                                        FB_Bacnet.StartStopCommand_139.bEnWrite := TRUE;
                                        FB_Bacnet.StartStopCommand_139.bVal := FALSE;
                                    13: 
                                        
                                        FB_Bacnet.StartStopCommand_140.bEnWrite := TRUE;
                                        FB_Bacnet.StartStopCommand_140.bVal := FALSE;
                                    14: 
                                        
                                        FB_Bacnet.StartStopCommand_141.bEnWrite := TRUE;
                                        FB_Bacnet.StartStopCommand_141.bVal := FALSE;
                                    15: 
                                        
                                        FB_Bacnet.StartStopCommand_142.bEnWrite := TRUE;
                                        FB_Bacnet.StartStopCommand_142.bVal := FALSE;
                                    16: 
                                        
                                        FB_Bacnet.StartStopCommand_143.bEnWrite := TRUE;
                                        FB_Bacnet.StartStopCommand_143.bVal := FALSE;
                                    17: 
                                        
                                        FB_Bacnet.StartStopCommand_144.bEnWrite := TRUE;
                                        FB_Bacnet.StartStopCommand_144.bVal := FALSE;
                                    18: 
                                        
                                        FB_Bacnet.StartStopCommand_145.bEnWrite := TRUE;
                                        FB_Bacnet.StartStopCommand_145.bVal := FALSE;
                                    19: 
                                        
                                        FB_Bacnet.StartStopCommand_146.bEnWrite := TRUE;
                                        FB_Bacnet.StartStopCommand_146.bVal := FALSE;
                                    20: 
                                        
                                        FB_Bacnet.StartStopCommand_147.bEnWrite := TRUE;
                                        FB_Bacnet.StartStopCommand_147.bVal := FALSE;
                                    21: 
                                        
                                        FB_Bacnet.StartStopCommand_148.bEnWrite := TRUE;
                                        FB_Bacnet.StartStopCommand_148.bVal := FALSE;
                                    22: 
                                        
                                        FB_Bacnet.StartStopCommand_149.bEnWrite := TRUE;
                                        FB_Bacnet.StartStopCommand_149.bVal := FALSE;
                                    23: 
                                        
                                        FB_Bacnet.StartStopCommand_226.bEnWrite := TRUE;
                                        FB_Bacnet.StartStopCommand_226.bVal := FALSE;
                                END_CASE
                            END_IF
                        END_FOR
                    END_IF
                END_IF
            END_IF

            // Weekend schedule
            IF currD = 0 OR currD = 6 THEN
                IF (wSchedWEHourStartF33_ <> wSchedWEHourEndF33_ OR wSchedWEMinStartF33_ <> wSchedWEMinEndF33_) THEN
                    // Schedule Unit ON
                    IF wSchedWEHourStartF33_ = currH AND wSchedWEMinStartF33_ = currM AND NOT bUnitTriggered THEN
                        bUnitTriggered := TRUE;
                        FOR i := 1 TO 23 DO
                            // Send command unit ON
                            IF bUnitF33_[i] THEN 
                                CASE i OF
                                    1: 
                                        
                                        FB_Bacnet.StartStopCommand_128.bEnWrite := TRUE;
                                        FB_Bacnet.StartStopCommand_128.bVal := TRUE;
                                    2: 
                                        
                                        FB_Bacnet.StartStopCommand_129.bEnWrite := TRUE;
                                        FB_Bacnet.StartStopCommand_129.bVal := TRUE;
                                    3: 
                                        
                                        FB_Bacnet.StartStopCommand_130.bEnWrite := TRUE;
                                        FB_Bacnet.StartStopCommand_130.bVal := TRUE;
                                    4: 
                                        
                                        FB_Bacnet.StartStopCommand_131.bEnWrite := TRUE;
                                        FB_Bacnet.StartStopCommand_131.bVal := TRUE;
                                    5: 
                                        
                                        FB_Bacnet.StartStopCommand_132.bEnWrite := TRUE;
                                        FB_Bacnet.StartStopCommand_132.bVal := TRUE;
                                    6: 
                                        
                                        FB_Bacnet.StartStopCommand_133.bEnWrite := TRUE;
                                        FB_Bacnet.StartStopCommand_133.bVal := TRUE;
                                    7: 
                                        
                                        FB_Bacnet.StartStopCommand_134.bEnWrite := TRUE;
                                        FB_Bacnet.StartStopCommand_134.bVal := TRUE;
                                    8: 
                                        
                                        FB_Bacnet.StartStopCommand_135.bEnWrite := TRUE;
                                        FB_Bacnet.StartStopCommand_135.bVal := TRUE;
                                    9: 
                                        
                                        FB_Bacnet.StartStopCommand_136.bEnWrite := TRUE;
                                        FB_Bacnet.StartStopCommand_136.bVal := TRUE;
                                    10: 
                                        
                                        FB_Bacnet.StartStopCommand_137.bEnWrite := TRUE;
                                        FB_Bacnet.StartStopCommand_137.bVal := TRUE;
                                    11: 
                                        
                                        FB_Bacnet.StartStopCommand_138.bEnWrite := TRUE;
                                        FB_Bacnet.StartStopCommand_138.bVal := TRUE;
                                    12: 
                                        
                                        FB_Bacnet.StartStopCommand_139.bEnWrite := TRUE;
                                        FB_Bacnet.StartStopCommand_139.bVal := TRUE;
                                    13: 
                                        
                                        FB_Bacnet.StartStopCommand_140.bEnWrite := TRUE;
                                        FB_Bacnet.StartStopCommand_140.bVal := TRUE;
                                    14: 
                                        
                                        FB_Bacnet.StartStopCommand_141.bEnWrite := TRUE;
                                        FB_Bacnet.StartStopCommand_141.bVal := TRUE;
                                    15: 
                                        
                                        FB_Bacnet.StartStopCommand_142.bEnWrite := TRUE;
                                        FB_Bacnet.StartStopCommand_142.bVal := TRUE;
                                    16: 
                                        
                                        FB_Bacnet.StartStopCommand_143.bEnWrite := TRUE;
                                        FB_Bacnet.StartStopCommand_143.bVal := TRUE;
                                    17: 
                                        
                                        FB_Bacnet.StartStopCommand_144.bEnWrite := TRUE;
                                        FB_Bacnet.StartStopCommand_144.bVal := TRUE;
                                    18: 
                                        
                                        FB_Bacnet.StartStopCommand_145.bEnWrite := TRUE;
                                        FB_Bacnet.StartStopCommand_145.bVal := TRUE;
                                    19: 
                                        
                                        FB_Bacnet.StartStopCommand_146.bEnWrite := TRUE;
                                        FB_Bacnet.StartStopCommand_146.bVal := TRUE;
                                    20: 
                                        
                                        FB_Bacnet.StartStopCommand_147.bEnWrite := TRUE;
                                        FB_Bacnet.StartStopCommand_147.bVal := TRUE;
                                    21: 
                                        
                                        FB_Bacnet.StartStopCommand_148.bEnWrite := TRUE;
                                        FB_Bacnet.StartStopCommand_148.bVal := TRUE;
                                    22: 
                                        
                                        FB_Bacnet.StartStopCommand_149.bEnWrite := TRUE;
                                        FB_Bacnet.StartStopCommand_149.bVal := TRUE;
                                    23: 
                                        
                                        FB_Bacnet.StartStopCommand_226.bEnWrite := TRUE;
                                        FB_Bacnet.StartStopCommand_226.bVal := TRUE;
                                END_CASE
                            END_IF
                        END_FOR
                    END_IF
                    // Schedule Unit OFF
                    IF wSchedWEHourEndF33_ = currH AND wSchedWEMinEndF33_ = currM AND NOT bUnitTriggered THEN
                        bUnitTriggered := TRUE;
                        FOR i := 1 TO 23 DO
                            // Send command unit OFF
                            IF bUnitF33_[i] THEN 
                                CASE i OF
                                    1: 
                                        
                                        FB_Bacnet.StartStopCommand_128.bEnWrite := TRUE;
                                        FB_Bacnet.StartStopCommand_128.bVal := FALSE;
                                    2: 
                                        
                                        FB_Bacnet.StartStopCommand_129.bEnWrite := TRUE;
                                        FB_Bacnet.StartStopCommand_129.bVal := FALSE;
                                    3: 
                                        
                                        FB_Bacnet.StartStopCommand_130.bEnWrite := TRUE;
                                        FB_Bacnet.StartStopCommand_130.bVal := FALSE;
                                    4: 
                                        
                                        FB_Bacnet.StartStopCommand_131.bEnWrite := TRUE;
                                        FB_Bacnet.StartStopCommand_131.bVal := FALSE;
                                    5: 
                                        
                                        FB_Bacnet.StartStopCommand_132.bEnWrite := TRUE;
                                        FB_Bacnet.StartStopCommand_132.bVal := FALSE;
                                    6: 
                                        
                                        FB_Bacnet.StartStopCommand_133.bEnWrite := TRUE;
                                        FB_Bacnet.StartStopCommand_133.bVal := FALSE;
                                    7: 
                                        
                                        FB_Bacnet.StartStopCommand_134.bEnWrite := TRUE;
                                        FB_Bacnet.StartStopCommand_134.bVal := FALSE;
                                    8: 
                                        
                                        FB_Bacnet.StartStopCommand_135.bEnWrite := TRUE;
                                        FB_Bacnet.StartStopCommand_135.bVal := FALSE;
                                    9: 
                                        
                                        FB_Bacnet.StartStopCommand_136.bEnWrite := TRUE;
                                        FB_Bacnet.StartStopCommand_136.bVal := FALSE;
                                    10: 
                                        
                                        FB_Bacnet.StartStopCommand_137.bEnWrite := TRUE;
                                        FB_Bacnet.StartStopCommand_137.bVal := FALSE;
                                    11: 
                                        
                                        FB_Bacnet.StartStopCommand_138.bEnWrite := TRUE;
                                        FB_Bacnet.StartStopCommand_138.bVal := FALSE;
                                    12: 
                                        
                                        FB_Bacnet.StartStopCommand_139.bEnWrite := TRUE;
                                        FB_Bacnet.StartStopCommand_139.bVal := FALSE;
                                    13: 
                                        
                                        FB_Bacnet.StartStopCommand_140.bEnWrite := TRUE;
                                        FB_Bacnet.StartStopCommand_140.bVal := FALSE;
                                    14: 
                                        
                                        FB_Bacnet.StartStopCommand_141.bEnWrite := TRUE;
                                        FB_Bacnet.StartStopCommand_141.bVal := FALSE;
                                    15: 
                                        
                                        FB_Bacnet.StartStopCommand_142.bEnWrite := TRUE;
                                        FB_Bacnet.StartStopCommand_142.bVal := FALSE;
                                    16: 
                                        
                                        FB_Bacnet.StartStopCommand_143.bEnWrite := TRUE;
                                        FB_Bacnet.StartStopCommand_143.bVal := FALSE;
                                    17: 
                                        
                                        FB_Bacnet.StartStopCommand_144.bEnWrite := TRUE;
                                        FB_Bacnet.StartStopCommand_144.bVal := FALSE;
                                    18: 
                                        
                                        FB_Bacnet.StartStopCommand_145.bEnWrite := TRUE;
                                        FB_Bacnet.StartStopCommand_145.bVal := FALSE;
                                    19: 
                                        
                                        FB_Bacnet.StartStopCommand_146.bEnWrite := TRUE;
                                        FB_Bacnet.StartStopCommand_146.bVal := FALSE;
                                    20: 
                                        
                                        FB_Bacnet.StartStopCommand_147.bEnWrite := TRUE;
                                        FB_Bacnet.StartStopCommand_147.bVal := FALSE;
                                    21: 
                                        
                                        FB_Bacnet.StartStopCommand_148.bEnWrite := TRUE;
                                        FB_Bacnet.StartStopCommand_148.bVal := FALSE;
                                    22: 
                                        
                                        FB_Bacnet.StartStopCommand_149.bEnWrite := TRUE;
                                        FB_Bacnet.StartStopCommand_149.bVal := FALSE;
                                    23: 
                                        
                                        FB_Bacnet.StartStopCommand_226.bEnWrite := TRUE;
                                        FB_Bacnet.StartStopCommand_226.bVal := FALSE;
                                END_CASE
                            END_IF
                        END_FOR
                    END_IF
                END_IF
            END_IF
        END_IF

END_FUNCTION_BLOCK

// ---- POUs/FB_Scheduler/FB_Scheduler_F35.TcPOU

    FUNCTION_BLOCK FB_Scheduler_F35
      VAR_INPUT
          currH : WORD;
          currM : WORD;
          currD : WORD;
      END_VAR
      VAR_IN_OUT
          FB_Bacnet : FB_BACnet_DAIKIN_MasterStation_III_No_8;
      END_VAR
      VAR
          i : INT;
          bUnitTriggered : BOOL := FALSE; // New flag to track execution
          prevMinute : WORD := 0;        // New variable to track the previous minute
      END_VAR
      VAR PERSISTENT
          //scheduler var
          bEnSchedF35_ : BOOL := FALSE;
          wSchedWDHourStartF35_ : WORD; 
          wSchedWDMinStartF35_ : WORD; 
          wSchedWEHourStartF35_ : WORD; 
          wSchedWEMinStartF35_ : WORD;
          wSchedWDHourEndF35_ : WORD;
          wSchedWDMinEndF35_ : WORD;
          wSchedWEHourEndF35_ : WORD;
          wSchedWEMinEndF35_ : WORD;
          //unit var
          bUnitF35_ : ARRAY [1..25] OF BOOL;
      END_VAR


// Reset trigger flag at minute change or at the exact scheduled time
IF currM <> prevMinute OR 
   (currH = wSchedWDHourStartF35_ AND currM = wSchedWDMinStartF35_) OR 
   (currH = wSchedWDHourEndF35_ AND currM = wSchedWDMinEndF35_) THEN
    bUnitTriggered := FALSE;
    prevMinute := currM;
END_IF

// Unit Schedule Enable
IF bEnSchedF35_ THEN
    // Weekday schedule
    IF currD >= 1 AND currD <= 5 THEN
        IF (wSchedWDHourStartF35_ <> wSchedWDHourEndF35_ OR wSchedWDMinStartF35_ <> wSchedWDMinEndF35_) THEN
            // Schedule Unit ON
            IF wSchedWDHourStartF35_ = currH AND wSchedWDMinStartF35_ = currM AND NOT bUnitTriggered THEN
                bUnitTriggered := TRUE;
                FOR i := 1 TO 25 DO
                    // Send command unit ON
                    IF bUnitF35_[i] THEN 
                        CASE i OF
                            1: 
                                FB_Bacnet.StartStopCommand_192.bEnWrite := TRUE;
                                FB_Bacnet.StartStopCommand_192.bVal := TRUE;
                            2: 
                                FB_Bacnet.StartStopCommand_193.bEnWrite := TRUE;
                                FB_Bacnet.StartStopCommand_193.bVal := TRUE;
                            3: 
                                FB_Bacnet.StartStopCommand_194.bEnWrite := TRUE;
                                FB_Bacnet.StartStopCommand_194.bVal := TRUE;
                            4: 
                                FB_Bacnet.StartStopCommand_195.bEnWrite := TRUE;
                                FB_Bacnet.StartStopCommand_195.bVal := TRUE;
                            5: 
                                FB_Bacnet.StartStopCommand_196.bEnWrite := TRUE;
                                FB_Bacnet.StartStopCommand_196.bVal := TRUE;
                            6: 
                                FB_Bacnet.StartStopCommand_197.bEnWrite := TRUE;
                                FB_Bacnet.StartStopCommand_197.bVal := TRUE;
                            7: 
                                FB_Bacnet.StartStopCommand_198.bEnWrite := TRUE;
                                FB_Bacnet.StartStopCommand_198.bVal := TRUE;
                            8: 
                                FB_Bacnet.StartStopCommand_199.bEnWrite := TRUE;
                                FB_Bacnet.StartStopCommand_199.bVal := TRUE;
                            9: 
                                FB_Bacnet.StartStopCommand_200.bEnWrite := TRUE;
                                FB_Bacnet.StartStopCommand_200.bVal := TRUE;
                            10: 
                                FB_Bacnet.StartStopCommand_201.bEnWrite := TRUE;
                                FB_Bacnet.StartStopCommand_201.bVal := TRUE;
                            11: 
                                FB_Bacnet.StartStopCommand_202.bEnWrite := TRUE;
                                FB_Bacnet.StartStopCommand_202.bVal := TRUE;
                            12: 
                                FB_Bacnet.StartStopCommand_203.bEnWrite := TRUE;
                                FB_Bacnet.StartStopCommand_203.bVal := TRUE;
                            13: 
                                FB_Bacnet.StartStopCommand_204.bEnWrite := TRUE;
                                FB_Bacnet.StartStopCommand_204.bVal := TRUE;
                            14: 
                                FB_Bacnet.StartStopCommand_205.bEnWrite := TRUE;
                                FB_Bacnet.StartStopCommand_205.bVal := TRUE;
                            15: 
                                FB_Bacnet.StartStopCommand_206.bEnWrite := TRUE;
                                FB_Bacnet.StartStopCommand_206.bVal := TRUE;
                            16: 
                                FB_Bacnet.StartStopCommand_207.bEnWrite := TRUE;
                                FB_Bacnet.StartStopCommand_207.bVal := TRUE;
                            17: 
                                FB_Bacnet.StartStopCommand_208.bEnWrite := TRUE;
                                FB_Bacnet.StartStopCommand_208.bVal := TRUE;
                            18: 
                                FB_Bacnet.StartStopCommand_209.bEnWrite := TRUE;
                                FB_Bacnet.StartStopCommand_209.bVal := TRUE;
                            19: 
                                FB_Bacnet.StartStopCommand_210.bEnWrite := TRUE;
                                FB_Bacnet.StartStopCommand_210.bVal := TRUE;
                            20: 
                                FB_Bacnet.StartStopCommand_211.bEnWrite := TRUE;
                                FB_Bacnet.StartStopCommand_211.bVal := TRUE;
                            21: 
                                FB_Bacnet.StartStopCommand_212.bEnWrite := TRUE;
                                FB_Bacnet.StartStopCommand_212.bVal := TRUE;
                            22: 
                                FB_Bacnet.StartStopCommand_213.bEnWrite := TRUE;
                                FB_Bacnet.StartStopCommand_213.bVal := TRUE;
                            23: 
                                //FB_Bacnet.StartStopCommand_242.bEnWrite := TRUE;
                                //FB_Bacnet.StartStopCommand_242.bVal := TRUE;
                            24: 
                                FB_Bacnet.StartStopCommand_243.bEnWrite := TRUE;
                                FB_Bacnet.StartStopCommand_243.bVal := TRUE;
                            25: 
                                FB_Bacnet.StartStopCommand_227.bEnWrite := TRUE;
                                FB_Bacnet.StartStopCommand_227.bVal := TRUE;
                        END_CASE
                    END_IF
                END_FOR
            END_IF
            // Schedule Unit OFF
            IF wSchedWDHourEndF35_ = currH AND wSchedWDMinEndF35_ = currM AND NOT bUnitTriggered THEN
                bUnitTriggered := TRUE;
                FOR i := 1 TO 25 DO
                    // Send command unit OFF
                    IF bUnitF35_[i] THEN 
                        CASE i OF
                            1: 
                                FB_Bacnet.StartStopCommand_192.bEnWrite := TRUE;
                                FB_Bacnet.StartStopCommand_192.bVal := FALSE;
                            2: 
                                FB_Bacnet.StartStopCommand_193.bEnWrite := TRUE;
                                FB_Bacnet.StartStopCommand_193.bVal := FALSE;
                            3: 
                                FB_Bacnet.StartStopCommand_194.bEnWrite := TRUE;
                                FB_Bacnet.StartStopCommand_194.bVal := FALSE;
                            4: 
                                FB_Bacnet.StartStopCommand_195.bEnWrite := TRUE;
                                FB_Bacnet.StartStopCommand_195.bVal := FALSE;
                            5: 
                                FB_Bacnet.StartStopCommand_196.bEnWrite := TRUE;
                                FB_Bacnet.StartStopCommand_196.bVal := FALSE;
                            6: 
                                FB_Bacnet.StartStopCommand_197.bEnWrite := TRUE;
                                FB_Bacnet.StartStopCommand_197.bVal := FALSE;
                            7: 
                                FB_Bacnet.StartStopCommand_198.bEnWrite := TRUE;
                                FB_Bacnet.StartStopCommand_198.bVal := FALSE;
                            8: 
                                FB_Bacnet.StartStopCommand_199.bEnWrite := TRUE;
                                FB_Bacnet.StartStopCommand_199.bVal := FALSE;
                            9: 
                                FB_Bacnet.StartStopCommand_200.bEnWrite := TRUE;
                                FB_Bacnet.StartStopCommand_200.bVal := FALSE;
                            10: 
                                FB_Bacnet.StartStopCommand_201.bEnWrite := TRUE;
                                FB_Bacnet.StartStopCommand_201.bVal := FALSE;
                            11: 
                                FB_Bacnet.StartStopCommand_202.bEnWrite := TRUE;
                                FB_Bacnet.StartStopCommand_202.bVal := FALSE;
                            12: 
                                FB_Bacnet.StartStopCommand_203.bEnWrite := TRUE;
                                FB_Bacnet.StartStopCommand_203.bVal := FALSE;
                            13: 
                                FB_Bacnet.StartStopCommand_204.bEnWrite := TRUE;
                                FB_Bacnet.StartStopCommand_204.bVal := FALSE;
                            14: 
                                FB_Bacnet.StartStopCommand_205.bEnWrite := TRUE;
                                FB_Bacnet.StartStopCommand_205.bVal := FALSE;
                            15: 
                                FB_Bacnet.StartStopCommand_206.bEnWrite := TRUE;
                                FB_Bacnet.StartStopCommand_206.bVal := FALSE;
                            16: 
                                FB_Bacnet.StartStopCommand_207.bEnWrite := TRUE;
                                FB_Bacnet.StartStopCommand_207.bVal := FALSE;
                            17: 
                                FB_Bacnet.StartStopCommand_208.bEnWrite := TRUE;
                                FB_Bacnet.StartStopCommand_208.bVal := FALSE;
                            18: 
                                FB_Bacnet.StartStopCommand_209.bEnWrite := TRUE;
                                FB_Bacnet.StartStopCommand_209.bVal := FALSE;
                            19: 
                                FB_Bacnet.StartStopCommand_210.bEnWrite := TRUE;
                                FB_Bacnet.StartStopCommand_210.bVal := FALSE;
                            20: 
                                FB_Bacnet.StartStopCommand_211.bEnWrite := TRUE;
                                FB_Bacnet.StartStopCommand_211.bVal := FALSE;
                            21: 
                                FB_Bacnet.StartStopCommand_212.bEnWrite := TRUE;
                                FB_Bacnet.StartStopCommand_212.bVal := FALSE;
                            22: 
                                FB_Bacnet.StartStopCommand_213.bEnWrite := TRUE;
                                FB_Bacnet.StartStopCommand_213.bVal := FALSE;
                            23: 
                                //FB_Bacnet.StartStopCommand_242.bEnWrite := TRUE;
                                //FB_Bacnet.StartStopCommand_242.bVal := FALSE;
                            24: 
                                FB_Bacnet.StartStopCommand_243.bEnWrite := TRUE;
                                FB_Bacnet.StartStopCommand_243.bVal := FALSE;
                            25: 
                                FB_Bacnet.StartStopCommand_227.bEnWrite := TRUE;
                                FB_Bacnet.StartStopCommand_227.bVal := FALSE;
                        END_CASE
                    END_IF
                END_FOR
            END_IF
        END_IF
    END_IF

    // Weekend schedule
    IF currD = 0 OR currD = 6 THEN
        IF (wSchedWEHourStartF35_ <> wSchedWEHourEndF35_ OR wSchedWEMinStartF35_ <> wSchedWEMinEndF35_) THEN
            // Schedule Unit ON
            IF wSchedWEHourStartF35_ = currH AND wSchedWEMinStartF35_ = currM AND NOT bUnitTriggered THEN
                bUnitTriggered := TRUE;
                FOR i := 1 TO 25 DO
                    // Send command unit ON
                    IF bUnitF35_[i] THEN 
                        CASE i OF
                            1: 
                                FB_Bacnet.StartStopCommand_192.bEnWrite := TRUE;
                                FB_Bacnet.StartStopCommand_192.bVal := TRUE;
                            2: 
                                FB_Bacnet.StartStopCommand_193.bEnWrite := TRUE;
                                FB_Bacnet.StartStopCommand_193.bVal := TRUE;
                            3: 
                                FB_Bacnet.StartStopCommand_194.bEnWrite := TRUE;
                                FB_Bacnet.StartStopCommand_194.bVal := TRUE;
                            4: 
                                FB_Bacnet.StartStopCommand_195.bEnWrite := TRUE;
                                FB_Bacnet.StartStopCommand_195.bVal := TRUE;
                            5: 
                                FB_Bacnet.StartStopCommand_196.bEnWrite := TRUE;
                                FB_Bacnet.StartStopCommand_196.bVal := TRUE;
                            6: 
                                FB_Bacnet.StartStopCommand_197.bEnWrite := TRUE;
                                FB_Bacnet.StartStopCommand_197.bVal := TRUE;
                            7: 
                                FB_Bacnet.StartStopCommand_198.bEnWrite := TRUE;
                                FB_Bacnet.StartStopCommand_198.bVal := TRUE;
                            8: 
                                FB_Bacnet.StartStopCommand_199.bEnWrite := TRUE;
                                FB_Bacnet.StartStopCommand_199.bVal := TRUE;
                            9: 
                                FB_Bacnet.StartStopCommand_200.bEnWrite := TRUE;
                                FB_Bacnet.StartStopCommand_200.bVal := TRUE;
                            10: 
                                FB_Bacnet.StartStopCommand_201.bEnWrite := TRUE;
                                FB_Bacnet.StartStopCommand_201.bVal := TRUE;
                            11: 
                                FB_Bacnet.StartStopCommand_202.bEnWrite := TRUE;
                                FB_Bacnet.StartStopCommand_202.bVal := TRUE;
                            12: 
                                FB_Bacnet.StartStopCommand_203.bEnWrite := TRUE;
                                FB_Bacnet.StartStopCommand_203.bVal := TRUE;
                            13: 
                                FB_Bacnet.StartStopCommand_204.bEnWrite := TRUE;
                                FB_Bacnet.StartStopCommand_204.bVal := TRUE;
                            14: 
                                FB_Bacnet.StartStopCommand_205.bEnWrite := TRUE;
                                FB_Bacnet.StartStopCommand_205.bVal := TRUE;
                            15: 
                                FB_Bacnet.StartStopCommand_206.bEnWrite := TRUE;
                                FB_Bacnet.StartStopCommand_206.bVal := TRUE;
                            16: 
                                FB_Bacnet.StartStopCommand_207.bEnWrite := TRUE;
                                FB_Bacnet.StartStopCommand_207.bVal := TRUE;
                            17: 
                                FB_Bacnet.StartStopCommand_208.bEnWrite := TRUE;
                                FB_Bacnet.StartStopCommand_208.bVal := TRUE;
                            18: 
                                FB_Bacnet.StartStopCommand_209.bEnWrite := TRUE;
                                FB_Bacnet.StartStopCommand_209.bVal := TRUE;
                            19: 
                                FB_Bacnet.StartStopCommand_210.bEnWrite := TRUE;
                                FB_Bacnet.StartStopCommand_210.bVal := TRUE;
                            20: 
                                FB_Bacnet.StartStopCommand_211.bEnWrite := TRUE;
                                FB_Bacnet.StartStopCommand_211.bVal := TRUE;
                            21: 
                                FB_Bacnet.StartStopCommand_212.bEnWrite := TRUE;
                                FB_Bacnet.StartStopCommand_212.bVal := TRUE;
                            22: 
                                FB_Bacnet.StartStopCommand_213.bEnWrite := TRUE;
                                FB_Bacnet.StartStopCommand_213.bVal := TRUE;
                            23: 
                                //FB_Bacnet.StartStopCommand_242.bEnWrite := TRUE;
                                //FB_Bacnet.StartStopCommand_242.bVal := TRUE;
                            24: 
                                FB_Bacnet.StartStopCommand_243.bEnWrite := TRUE;
                                FB_Bacnet.StartStopCommand_243.bVal := TRUE;
                            25: 
                                FB_Bacnet.StartStopCommand_227.bEnWrite := TRUE;
                                FB_Bacnet.StartStopCommand_227.bVal := TRUE;
                        END_CASE
                    END_IF
                END_FOR        
            END_IF
            // Schedule Unit OFF
            IF wSchedWEHourEndF35_ = currH AND wSchedWEMinEndF35_ = currM AND NOT bUnitTriggered THEN
                bUnitTriggered := TRUE;
                FOR i := 1 TO 25 DO
                    // Send command unit OFF
                    IF bUnitF35_[i] THEN 
                        CASE i OF
                            1: 
                                FB_Bacnet.StartStopCommand_192.bEnWrite := TRUE;
                                FB_Bacnet.StartStopCommand_192.bVal := FALSE;
                            2: 
                                FB_Bacnet.StartStopCommand_193.bEnWrite := TRUE;
                                FB_Bacnet.StartStopCommand_193.bVal := FALSE;
                            3: 
                                FB_Bacnet.StartStopCommand_194.bEnWrite := TRUE;
                                FB_Bacnet.StartStopCommand_194.bVal := FALSE;
                            4: 
                                FB_Bacnet.StartStopCommand_195.bEnWrite := TRUE;
                                FB_Bacnet.StartStopCommand_195.bVal := FALSE;
                            5: 
                                FB_Bacnet.StartStopCommand_196.bEnWrite := TRUE;
                                FB_Bacnet.StartStopCommand_196.bVal := FALSE;
                            6: 
                                FB_Bacnet.StartStopCommand_197.bEnWrite := TRUE;
                                FB_Bacnet.StartStopCommand_197.bVal := FALSE;
                            7: 
                                FB_Bacnet.StartStopCommand_198.bEnWrite := TRUE;
                                FB_Bacnet.StartStopCommand_198.bVal := FALSE;
                            8: 
                                FB_Bacnet.StartStopCommand_199.bEnWrite := TRUE;
                                FB_Bacnet.StartStopCommand_199.bVal := FALSE;
                            9: 
                                FB_Bacnet.StartStopCommand_200.bEnWrite := TRUE;
                                FB_Bacnet.StartStopCommand_200.bVal := FALSE;
                            10: 
                                FB_Bacnet.StartStopCommand_201.bEnWrite := TRUE;
                                FB_Bacnet.StartStopCommand_201.bVal := FALSE;
                            11: 
                                FB_Bacnet.StartStopCommand_202.bEnWrite := TRUE;
                                FB_Bacnet.StartStopCommand_202.bVal := FALSE;
                            12: 
                                FB_Bacnet.StartStopCommand_203.bEnWrite := TRUE;
                                FB_Bacnet.StartStopCommand_203.bVal := FALSE;
                            13: 
                                FB_Bacnet.StartStopCommand_204.bEnWrite := TRUE;
                                FB_Bacnet.StartStopCommand_204.bVal := FALSE;
                            14: 
                                FB_Bacnet.StartStopCommand_205.bEnWrite := TRUE;
                                FB_Bacnet.StartStopCommand_205.bVal := FALSE;
                            15: 
                                FB_Bacnet.StartStopCommand_206.bEnWrite := TRUE;
                                FB_Bacnet.StartStopCommand_206.bVal := FALSE;
                            16: 
                                FB_Bacnet.StartStopCommand_207.bEnWrite := TRUE;
                                FB_Bacnet.StartStopCommand_207.bVal := FALSE;
                            17: 
                                FB_Bacnet.StartStopCommand_208.bEnWrite := TRUE;
                                FB_Bacnet.StartStopCommand_208.bVal := FALSE;
                            18: 
                                FB_Bacnet.StartStopCommand_209.bEnWrite := TRUE;
                                FB_Bacnet.StartStopCommand_209.bVal := FALSE;
                            19: 
                                FB_Bacnet.StartStopCommand_210.bEnWrite := TRUE;
                                FB_Bacnet.StartStopCommand_210.bVal := FALSE;
                            20: 
                                FB_Bacnet.StartStopCommand_211.bEnWrite := TRUE;
                                FB_Bacnet.StartStopCommand_211.bVal := FALSE;
                            21: 
                                FB_Bacnet.StartStopCommand_212.bEnWrite := TRUE;
                                FB_Bacnet.StartStopCommand_212.bVal := FALSE;
                            22: 
                                FB_Bacnet.StartStopCommand_213.bEnWrite := TRUE;
                                FB_Bacnet.StartStopCommand_213.bVal := FALSE;
                            23: 
                                //FB_Bacnet.StartStopCommand_242.bEnWrite := TRUE;
                                //FB_Bacnet.StartStopCommand_242.bVal := FALSE;
                            24: 
                                FB_Bacnet.StartStopCommand_243.bEnWrite := TRUE;
                                FB_Bacnet.StartStopCommand_243.bVal := FALSE;
                            25: 
                                FB_Bacnet.StartStopCommand_227.bEnWrite := TRUE;
                                FB_Bacnet.StartStopCommand_227.bVal := FALSE;
                        END_CASE
                    END_IF
                END_FOR
            END_IF
        END_IF
    END_IF
END_IF

END_FUNCTION_BLOCK

// ---- POUs/FB_Scheduler/FB_Scheduler_F36.TcPOU

      FUNCTION_BLOCK FB_Scheduler_F36
      VAR_INPUT
          currH : WORD;
          currM : WORD;
          currD : WORD;
      END_VAR
      VAR_IN_OUT
          FB_Bacnet : FB_BACnet_DAIKIN_MasterStation_III_No_9;
      END_VAR
      VAR
          i : INT;
          bUnitTriggered : BOOL := FALSE; // New flag to track execution
          prevMinute : WORD := 0;        // New variable to track the previous minute
      END_VAR
      VAR PERSISTENT
          //scheduler var
          bEnSchedF36_ : BOOL := FALSE;
          wSchedWDHourStartF36_ : WORD; 
          wSchedWDMinStartF36_ : WORD; 
          wSchedWEHourStartF36_ : WORD; 
          wSchedWEMinStartF36_ : WORD;
          wSchedWDHourEndF36_ : WORD;
          wSchedWDMinEndF36_ : WORD;
          wSchedWEHourEndF36_ : WORD;
          wSchedWEMinEndF36_ : WORD;
          //unit var
          bUnitF36_ : ARRAY [1..23] OF BOOL;
      END_VAR


        // Reset trigger flag at minute change or at the exact scheduled time
        IF currM <> prevMinute OR 
           (currH = wSchedWDHourStartF36_ AND currM = wSchedWDMinStartF36_) OR 
           (currH = wSchedWDHourEndF36_ AND currM = wSchedWDMinEndF36_) THEN
            bUnitTriggered := FALSE;
            prevMinute := currM;
        END_IF

        // Unit Schedule Enable
        IF bEnSchedF36_ THEN
            // Weekday schedule
            IF currD >= 1 AND currD <= 5 THEN
                IF (wSchedWDHourStartF36_ <> wSchedWDHourEndF36_ OR wSchedWDMinStartF36_ <> wSchedWDMinEndF36_) THEN
                    // Schedule Unit ON
                    IF wSchedWDHourStartF36_ = currH AND wSchedWDMinStartF36_ = currM AND NOT bUnitTriggered THEN
                        bUnitTriggered := TRUE;
                        FOR i := 1 TO 23 DO
                            // Send command unit ON
                            IF bUnitF36_[i] THEN 
                                CASE i OF
                                    1: 
                                        
                                        FB_Bacnet.StartStopCommand_000.bEnWrite := TRUE;
                                        FB_Bacnet.StartStopCommand_000.bVal := TRUE;
                                    2: 
                                        
                                        FB_Bacnet.StartStopCommand_001.bEnWrite := TRUE;
                                        FB_Bacnet.StartStopCommand_001.bVal := TRUE;
                                    3: 
                                        
                                        FB_Bacnet.StartStopCommand_002.bEnWrite := TRUE;
                                        FB_Bacnet.StartStopCommand_002.bVal := TRUE;
                                    4: 
                                        
                                        FB_Bacnet.StartStopCommand_003.bEnWrite := TRUE;
                                        FB_Bacnet.StartStopCommand_003.bVal := TRUE;
                                    5: 
                                        
                                        FB_Bacnet.StartStopCommand_004.bEnWrite := TRUE;
                                        FB_Bacnet.StartStopCommand_004.bVal := TRUE;
                                    6: 
                                        
                                        FB_Bacnet.StartStopCommand_005.bEnWrite := TRUE;
                                        FB_Bacnet.StartStopCommand_005.bVal := TRUE;
                                    7: 
                                        
                                        FB_Bacnet.StartStopCommand_006.bEnWrite := TRUE;
                                        FB_Bacnet.StartStopCommand_006.bVal := TRUE;
                                    8: 
                                        
                                        FB_Bacnet.StartStopCommand_007.bEnWrite := TRUE;
                                        FB_Bacnet.StartStopCommand_007.bVal := TRUE;
                                    9: 
                                        
                                        FB_Bacnet.StartStopCommand_008.bEnWrite := TRUE;
                                        FB_Bacnet.StartStopCommand_008.bVal := TRUE;
                                    10: 
                                        
                                        FB_Bacnet.StartStopCommand_009.bEnWrite := TRUE;
                                        FB_Bacnet.StartStopCommand_009.bVal := TRUE;
                                    11: 
                                        
                                        FB_Bacnet.StartStopCommand_010.bEnWrite := TRUE;
                                        FB_Bacnet.StartStopCommand_010.bVal := TRUE;
                                    12: 
                                        
                                        FB_Bacnet.StartStopCommand_011.bEnWrite := TRUE;
                                        FB_Bacnet.StartStopCommand_011.bVal := TRUE;
                                    13: 
                                        
                                        FB_Bacnet.StartStopCommand_012.bEnWrite := TRUE;
                                        FB_Bacnet.StartStopCommand_012.bVal := TRUE;
                                    14: 
                                        
                                        FB_Bacnet.StartStopCommand_013.bEnWrite := TRUE;
                                        FB_Bacnet.StartStopCommand_013.bVal := TRUE;
                                    15: 
                                        
                                        FB_Bacnet.StartStopCommand_014.bEnWrite := TRUE;
                                        FB_Bacnet.StartStopCommand_014.bVal := TRUE;
                                    16: 
                                        
                                        FB_Bacnet.StartStopCommand_015.bEnWrite := TRUE;
                                        FB_Bacnet.StartStopCommand_015.bVal := TRUE;
                                    17: 
                                        
                                        FB_Bacnet.StartStopCommand_016.bEnWrite := TRUE;
                                        FB_Bacnet.StartStopCommand_016.bVal := TRUE;
                                    18: 
                                        
                                        FB_Bacnet.StartStopCommand_017.bEnWrite := TRUE;
                                        FB_Bacnet.StartStopCommand_017.bVal := TRUE;
                                    19: 
                                        
                                        FB_Bacnet.StartStopCommand_018.bEnWrite := TRUE;
                                        FB_Bacnet.StartStopCommand_018.bVal := TRUE;
                                    20: 
                                        
                                        FB_Bacnet.StartStopCommand_019.bEnWrite := TRUE;
                                        FB_Bacnet.StartStopCommand_019.bVal := TRUE;
                                    21: 
                                        
                                        FB_Bacnet.StartStopCommand_020.bEnWrite := TRUE;
                                        FB_Bacnet.StartStopCommand_020.bVal := TRUE;
                                    22: 
                                        
                                        FB_Bacnet.StartStopCommand_021.bEnWrite := TRUE;
                                        FB_Bacnet.StartStopCommand_021.bVal := TRUE;
                                    23: 
                                        
                                        FB_Bacnet.StartStopCommand_224.bEnWrite := TRUE;
                                        FB_Bacnet.StartStopCommand_224.bVal := TRUE;
                                END_CASE
                            END_IF
                        END_FOR
                    END_IF
                    // Schedule Unit OFF
                    IF wSchedWDHourEndF36_ = currH AND wSchedWDMinEndF36_ = currM AND NOT bUnitTriggered THEN
                        bUnitTriggered := TRUE;
                        FOR i := 1 TO 23 DO
                            // Send command unit OFF
                            IF bUnitF36_[i] THEN 
                                CASE i OF
                                    1: 
                                        
                                        FB_Bacnet.StartStopCommand_000.bEnWrite := TRUE;
                                        FB_Bacnet.StartStopCommand_000.bVal := FALSE;
                                    2: 
                                        
                                        FB_Bacnet.StartStopCommand_001.bEnWrite := TRUE;
                                        FB_Bacnet.StartStopCommand_001.bVal := FALSE;
                                    3: 
                                        
                                        FB_Bacnet.StartStopCommand_002.bEnWrite := TRUE;
                                        FB_Bacnet.StartStopCommand_002.bVal := FALSE;
                                    4: 
                                        
                                        FB_Bacnet.StartStopCommand_003.bEnWrite := TRUE;
                                        FB_Bacnet.StartStopCommand_003.bVal := FALSE;
                                    5: 
                                        
                                        FB_Bacnet.StartStopCommand_004.bEnWrite := TRUE;
                                        FB_Bacnet.StartStopCommand_004.bVal := FALSE;
                                    6: 
                                        
                                        FB_Bacnet.StartStopCommand_005.bEnWrite := TRUE;
                                        FB_Bacnet.StartStopCommand_005.bVal := FALSE;
                                    7: 
                                        
                                        FB_Bacnet.StartStopCommand_006.bEnWrite := TRUE;
                                        FB_Bacnet.StartStopCommand_006.bVal := FALSE;
                                    8: 
                                        
                                        FB_Bacnet.StartStopCommand_007.bEnWrite := TRUE;
                                        FB_Bacnet.StartStopCommand_007.bVal := FALSE;
                                    9: 
                                        
                                        FB_Bacnet.StartStopCommand_008.bEnWrite := TRUE;
                                        FB_Bacnet.StartStopCommand_008.bVal := FALSE;
                                    10: 
                                        
                                        FB_Bacnet.StartStopCommand_009.bEnWrite := TRUE;
                                        FB_Bacnet.StartStopCommand_009.bVal := FALSE;
                                    11: 
                                        
                                        FB_Bacnet.StartStopCommand_010.bEnWrite := TRUE;
                                        FB_Bacnet.StartStopCommand_010.bVal := FALSE;
                                    12: 
                                        
                                        FB_Bacnet.StartStopCommand_011.bEnWrite := TRUE;
                                        FB_Bacnet.StartStopCommand_011.bVal := FALSE;
                                    13: 
                                        
                                        FB_Bacnet.StartStopCommand_012.bEnWrite := TRUE;
                                        FB_Bacnet.StartStopCommand_012.bVal := FALSE;
                                    14: 
                                        
                                        FB_Bacnet.StartStopCommand_013.bEnWrite := TRUE;
                                        FB_Bacnet.StartStopCommand_013.bVal := FALSE;
                                    15: 
                                        
                                        FB_Bacnet.StartStopCommand_014.bEnWrite := TRUE;
                                        FB_Bacnet.StartStopCommand_014.bVal := FALSE;
                                    16: 
                                        
                                        FB_Bacnet.StartStopCommand_015.bEnWrite := TRUE;
                                        FB_Bacnet.StartStopCommand_015.bVal := FALSE;
                                    17: 
                                        
                                        FB_Bacnet.StartStopCommand_016.bEnWrite := TRUE;
                                        FB_Bacnet.StartStopCommand_016.bVal := FALSE;
                                    18: 
                                        
                                        FB_Bacnet.StartStopCommand_017.bEnWrite := TRUE;
                                        FB_Bacnet.StartStopCommand_017.bVal := FALSE;
                                    19: 
                                        
                                        FB_Bacnet.StartStopCommand_018.bEnWrite := TRUE;
                                        FB_Bacnet.StartStopCommand_018.bVal := FALSE;
                                    20: 
                                        
                                        FB_Bacnet.StartStopCommand_019.bEnWrite := TRUE;
                                        FB_Bacnet.StartStopCommand_019.bVal := FALSE;
                                    21: 
                                        
                                        FB_Bacnet.StartStopCommand_020.bEnWrite := TRUE;
                                        FB_Bacnet.StartStopCommand_020.bVal := FALSE;
                                    22: 
                                        
                                        FB_Bacnet.StartStopCommand_021.bEnWrite := TRUE;
                                        FB_Bacnet.StartStopCommand_021.bVal := FALSE;
                                    23: 
                                        
                                        FB_Bacnet.StartStopCommand_224.bEnWrite := TRUE;
                                        FB_Bacnet.StartStopCommand_224.bVal := FALSE;
                                END_CASE
                            END_IF
                        END_FOR
                    END_IF
                END_IF
            END_IF

            // Weekend schedule
            IF currD = 0 OR currD = 6 THEN
                IF (wSchedWEHourStartF36_ <> wSchedWEHourEndF36_ OR wSchedWEMinStartF36_ <> wSchedWEMinEndF36_) THEN
                    // Schedule Unit ON
                    IF wSchedWEHourStartF36_ = currH AND wSchedWEMinStartF36_ = currM AND NOT bUnitTriggered THEN
                        bUnitTriggered := TRUE;
                        FOR i := 1 TO 23 DO
                            // Send command unit ON
                            IF bUnitF36_[i] THEN 
                                CASE i OF
                                    1: 
                                        
                                        FB_Bacnet.StartStopCommand_000.bEnWrite := TRUE;
                                        FB_Bacnet.StartStopCommand_000.bVal := TRUE;
                                    2: 
                                        
                                        FB_Bacnet.StartStopCommand_001.bEnWrite := TRUE;
                                        FB_Bacnet.StartStopCommand_001.bVal := TRUE;
                                    3: 
                                        
                                        FB_Bacnet.StartStopCommand_002.bEnWrite := TRUE;
                                        FB_Bacnet.StartStopCommand_002.bVal := TRUE;
                                    4: 
                                        
                                        FB_Bacnet.StartStopCommand_003.bEnWrite := TRUE;
                                        FB_Bacnet.StartStopCommand_003.bVal := TRUE;
                                    5: 
                                        
                                        FB_Bacnet.StartStopCommand_004.bEnWrite := TRUE;
                                        FB_Bacnet.StartStopCommand_004.bVal := TRUE;
                                    6: 
                                        
                                        FB_Bacnet.StartStopCommand_005.bEnWrite := TRUE;
                                        FB_Bacnet.StartStopCommand_005.bVal := TRUE;
                                    7: 
                                        
                                        FB_Bacnet.StartStopCommand_006.bEnWrite := TRUE;
                                        FB_Bacnet.StartStopCommand_006.bVal := TRUE;
                                    8: 
                                        
                                        FB_Bacnet.StartStopCommand_007.bEnWrite := TRUE;
                                        FB_Bacnet.StartStopCommand_007.bVal := TRUE;
                                    9: 
                                        
                                        FB_Bacnet.StartStopCommand_008.bEnWrite := TRUE;
                                        FB_Bacnet.StartStopCommand_008.bVal := TRUE;
                                    10: 
                                        
                                        FB_Bacnet.StartStopCommand_009.bEnWrite := TRUE;
                                        FB_Bacnet.StartStopCommand_009.bVal := TRUE;
                                    11: 
                                        
                                        FB_Bacnet.StartStopCommand_010.bEnWrite := TRUE;
                                        FB_Bacnet.StartStopCommand_010.bVal := TRUE;
                                    12: 
                                        
                                        FB_Bacnet.StartStopCommand_011.bEnWrite := TRUE;
                                        FB_Bacnet.StartStopCommand_011.bVal := TRUE;
                                    13: 
                                        
                                        FB_Bacnet.StartStopCommand_012.bEnWrite := TRUE;
                                        FB_Bacnet.StartStopCommand_012.bVal := TRUE;
                                    14: 
                                        
                                        FB_Bacnet.StartStopCommand_013.bEnWrite := TRUE;
                                        FB_Bacnet.StartStopCommand_013.bVal := TRUE;
                                    15: 
                                        
                                        FB_Bacnet.StartStopCommand_014.bEnWrite := TRUE;
                                        FB_Bacnet.StartStopCommand_014.bVal := TRUE;
                                    16: 
                                        
                                        FB_Bacnet.StartStopCommand_015.bEnWrite := TRUE;
                                        FB_Bacnet.StartStopCommand_015.bVal := TRUE;
                                    17: 
                                        
                                        FB_Bacnet.StartStopCommand_016.bEnWrite := TRUE;
                                        FB_Bacnet.StartStopCommand_016.bVal := TRUE;
                                    18: 
                                        
                                        FB_Bacnet.StartStopCommand_017.bEnWrite := TRUE;
                                        FB_Bacnet.StartStopCommand_017.bVal := TRUE;
                                    19: 
                                        
                                        FB_Bacnet.StartStopCommand_018.bEnWrite := TRUE;
                                        FB_Bacnet.StartStopCommand_018.bVal := TRUE;
                                    20: 
                                        
                                        FB_Bacnet.StartStopCommand_019.bEnWrite := TRUE;
                                        FB_Bacnet.StartStopCommand_019.bVal := TRUE;
                                    21: 
                                        
                                        FB_Bacnet.StartStopCommand_020.bEnWrite := TRUE;
                                        FB_Bacnet.StartStopCommand_020.bVal := TRUE;
                                    22: 
                                        
                                        FB_Bacnet.StartStopCommand_021.bEnWrite := TRUE;
                                        FB_Bacnet.StartStopCommand_021.bVal := TRUE;
                                    23: 
                                        
                                        FB_Bacnet.StartStopCommand_224.bEnWrite := TRUE;
                                        FB_Bacnet.StartStopCommand_224.bVal := TRUE;
                                END_CASE
                            END_IF
                        END_FOR
                    END_IF
                    // Schedule Unit OFF
                    IF wSchedWEHourEndF36_ = currH AND wSchedWEMinEndF36_ = currM AND NOT bUnitTriggered THEN
                        bUnitTriggered := TRUE;
                        FOR i := 1 TO 23 DO
                            // Send command unit OFF
                            IF bUnitF36_[i] THEN 
                                CASE i OF
                                    1: 
                                        
                                        FB_Bacnet.StartStopCommand_000.bEnWrite := TRUE;
                                        FB_Bacnet.StartStopCommand_000.bVal := FALSE;
                                    2: 
                                        
                                        FB_Bacnet.StartStopCommand_001.bEnWrite := TRUE;
                                        FB_Bacnet.StartStopCommand_001.bVal := FALSE;
                                    3: 
                                        
                                        FB_Bacnet.StartStopCommand_002.bEnWrite := TRUE;
                                        FB_Bacnet.StartStopCommand_002.bVal := FALSE;
                                    4: 
                                        
                                        FB_Bacnet.StartStopCommand_003.bEnWrite := TRUE;
                                        FB_Bacnet.StartStopCommand_003.bVal := FALSE;
                                    5: 
                                        
                                        FB_Bacnet.StartStopCommand_004.bEnWrite := TRUE;
                                        FB_Bacnet.StartStopCommand_004.bVal := FALSE;
                                    6: 
                                        
                                        FB_Bacnet.StartStopCommand_005.bEnWrite := TRUE;
                                        FB_Bacnet.StartStopCommand_005.bVal := FALSE;
                                    7: 
                                        
                                        FB_Bacnet.StartStopCommand_006.bEnWrite := TRUE;
                                        FB_Bacnet.StartStopCommand_006.bVal := FALSE;
                                    8: 
                                        
                                        FB_Bacnet.StartStopCommand_007.bEnWrite := TRUE;
                                        FB_Bacnet.StartStopCommand_007.bVal := FALSE;
                                    9: 
                                        
                                        FB_Bacnet.StartStopCommand_008.bEnWrite := TRUE;
                                        FB_Bacnet.StartStopCommand_008.bVal := FALSE;
                                    10: 
                                        
                                        FB_Bacnet.StartStopCommand_009.bEnWrite := TRUE;
                                        FB_Bacnet.StartStopCommand_009.bVal := FALSE;
                                    11: 
                                        
                                        FB_Bacnet.StartStopCommand_010.bEnWrite := TRUE;
                                        FB_Bacnet.StartStopCommand_010.bVal := FALSE;
                                    12: 
                                        
                                        FB_Bacnet.StartStopCommand_011.bEnWrite := TRUE;
                                        FB_Bacnet.StartStopCommand_011.bVal := FALSE;
                                    13: 
                                        
                                        FB_Bacnet.StartStopCommand_012.bEnWrite := TRUE;
                                        FB_Bacnet.StartStopCommand_012.bVal := FALSE;
                                    14: 
                                        
                                        FB_Bacnet.StartStopCommand_013.bEnWrite := TRUE;
                                        FB_Bacnet.StartStopCommand_013.bVal := FALSE;
                                    15: 
                                        
                                        FB_Bacnet.StartStopCommand_014.bEnWrite := TRUE;
                                        FB_Bacnet.StartStopCommand_014.bVal := FALSE;
                                    16: 
                                        
                                        FB_Bacnet.StartStopCommand_015.bEnWrite := TRUE;
                                        FB_Bacnet.StartStopCommand_015.bVal := FALSE;
                                    17: 
                                        
                                        FB_Bacnet.StartStopCommand_016.bEnWrite := TRUE;
                                        FB_Bacnet.StartStopCommand_016.bVal := FALSE;
                                    18: 
                                        
                                        FB_Bacnet.StartStopCommand_017.bEnWrite := TRUE;
                                        FB_Bacnet.StartStopCommand_017.bVal := FALSE;
                                    19: 
                                        
                                        FB_Bacnet.StartStopCommand_018.bEnWrite := TRUE;
                                        FB_Bacnet.StartStopCommand_018.bVal := FALSE;
                                    20: 
                                        
                                        FB_Bacnet.StartStopCommand_019.bEnWrite := TRUE;
                                        FB_Bacnet.StartStopCommand_019.bVal := FALSE;
                                    21: 
                                        
                                        FB_Bacnet.StartStopCommand_020.bEnWrite := TRUE;
                                        FB_Bacnet.StartStopCommand_020.bVal := FALSE;
                                    22: 
                                        
                                        FB_Bacnet.StartStopCommand_021.bEnWrite := TRUE;
                                        FB_Bacnet.StartStopCommand_021.bVal := FALSE;
                                    23: 
                                        
                                        FB_Bacnet.StartStopCommand_224.bEnWrite := TRUE;
                                        FB_Bacnet.StartStopCommand_224.bVal := FALSE;
                                END_CASE
                            END_IF
                        END_FOR
                    END_IF
                END_IF
            END_IF
        END_IF

END_FUNCTION_BLOCK

// ---- POUs/FB_Scheduler/FB_Scheduler_F37.TcPOU

      FUNCTION_BLOCK FB_Scheduler_F37
      VAR_INPUT
          currH : WORD;
          currM : WORD;
          currD : WORD;
      END_VAR
      VAR_IN_OUT
          FB_Bacnet : FB_BACnet_DAIKIN_MasterStation_III_No_9;
      END_VAR
      VAR
          i : INT;
          bUnitTriggered : BOOL := FALSE; // New flag to track execution
          prevMinute : WORD := 0;        // New variable to track the previous minute
      END_VAR
      VAR PERSISTENT
          //scheduler var
          bEnSchedF37_ : BOOL := FALSE;
          wSchedWDHourStartF37_ : WORD; 
          wSchedWDMinStartF37_ : WORD; 
          wSchedWEHourStartF37_ : WORD; 
          wSchedWEMinStartF37_ : WORD;
          wSchedWDHourEndF37_ : WORD;
          wSchedWDMinEndF37_ : WORD;
          wSchedWEHourEndF37_ : WORD;
          wSchedWEMinEndF37_ : WORD;
          //unit var
          bUnitF37_ : ARRAY [1..23] OF BOOL;
      END_VAR


        // Reset trigger flag at minute change or at the exact scheduled time
        IF currM <> prevMinute OR 
           (currH = wSchedWDHourStartF37_ AND currM = wSchedWDMinStartF37_) OR 
           (currH = wSchedWDHourEndF37_ AND currM = wSchedWDMinEndF37_) THEN
            bUnitTriggered := FALSE;
            prevMinute := currM;
        END_IF

        // Unit Schedule Enable
        IF bEnSchedF37_ THEN
            // Weekday schedule
            IF currD >= 1 AND currD <= 5 THEN
                IF (wSchedWDHourStartF37_ <> wSchedWDHourEndF37_ OR wSchedWDMinStartF37_ <> wSchedWDMinEndF37_) THEN
                    // Schedule Unit ON
                    IF wSchedWDHourStartF37_ = currH AND wSchedWDMinStartF37_ = currM AND NOT bUnitTriggered THEN
                        bUnitTriggered := TRUE;
                        FOR i := 1 TO 23 DO
                            // Send command unit ON
                            IF bUnitF37_[i] THEN 
                                CASE i OF
                                    1: 
                                        
                                        FB_Bacnet.StartStopCommand_064.bEnWrite := TRUE;
                                        FB_Bacnet.StartStopCommand_064.bVal := TRUE;
                                    2: 
                                        
                                        FB_Bacnet.StartStopCommand_065.bEnWrite := TRUE;
                                        FB_Bacnet.StartStopCommand_065.bVal := TRUE;
                                    3: 
                                        
                                        FB_Bacnet.StartStopCommand_066.bEnWrite := TRUE;
                                        FB_Bacnet.StartStopCommand_066.bVal := TRUE;
                                    4: 
                                        
                                        FB_Bacnet.StartStopCommand_067.bEnWrite := TRUE;
                                        FB_Bacnet.StartStopCommand_067.bVal := TRUE;
                                    5: 
                                        
                                        FB_Bacnet.StartStopCommand_068.bEnWrite := TRUE;
                                        FB_Bacnet.StartStopCommand_068.bVal := TRUE;
                                    6: 
                                        
                                        FB_Bacnet.StartStopCommand_069.bEnWrite := TRUE;
                                        FB_Bacnet.StartStopCommand_069.bVal := TRUE;
                                    7: 
                                        
                                        FB_Bacnet.StartStopCommand_070.bEnWrite := TRUE;
                                        FB_Bacnet.StartStopCommand_070.bVal := TRUE;
                                    8: 
                                        
                                        FB_Bacnet.StartStopCommand_071.bEnWrite := TRUE;
                                        FB_Bacnet.StartStopCommand_071.bVal := TRUE;
                                    9: 
                                        
                                        FB_Bacnet.StartStopCommand_072.bEnWrite := TRUE;
                                        FB_Bacnet.StartStopCommand_072.bVal := TRUE;
                                    10: 
                                        
                                        FB_Bacnet.StartStopCommand_073.bEnWrite := TRUE;
                                        FB_Bacnet.StartStopCommand_073.bVal := TRUE;
                                    11: 
                                        
                                        FB_Bacnet.StartStopCommand_074.bEnWrite := TRUE;
                                        FB_Bacnet.StartStopCommand_074.bVal := TRUE;
                                    12: 
                                        
                                        FB_Bacnet.StartStopCommand_075.bEnWrite := TRUE;
                                        FB_Bacnet.StartStopCommand_075.bVal := TRUE;
                                    13: 
                                        
                                        FB_Bacnet.StartStopCommand_076.bEnWrite := TRUE;
                                        FB_Bacnet.StartStopCommand_076.bVal := TRUE;
                                    14: 
                                        
                                        FB_Bacnet.StartStopCommand_077.bEnWrite := TRUE;
                                        FB_Bacnet.StartStopCommand_077.bVal := TRUE;
                                    15: 
                                        
                                        FB_Bacnet.StartStopCommand_078.bEnWrite := TRUE;
                                        FB_Bacnet.StartStopCommand_078.bVal := TRUE;
                                    16: 
                                        
                                        FB_Bacnet.StartStopCommand_079.bEnWrite := TRUE;
                                        FB_Bacnet.StartStopCommand_079.bVal := TRUE;
                                    17: 
                                        
                                        FB_Bacnet.StartStopCommand_080.bEnWrite := TRUE;
                                        FB_Bacnet.StartStopCommand_080.bVal := TRUE;
                                    18: 
                                        
                                        FB_Bacnet.StartStopCommand_081.bEnWrite := TRUE;
                                        FB_Bacnet.StartStopCommand_081.bVal := TRUE;
                                    19: 
                                        
                                        FB_Bacnet.StartStopCommand_082.bEnWrite := TRUE;
                                        FB_Bacnet.StartStopCommand_082.bVal := TRUE;
                                    20: 
                                        
                                        FB_Bacnet.StartStopCommand_083.bEnWrite := TRUE;
                                        FB_Bacnet.StartStopCommand_083.bVal := TRUE;
                                    21: 
                                        
                                        FB_Bacnet.StartStopCommand_084.bEnWrite := TRUE;
                                        FB_Bacnet.StartStopCommand_084.bVal := TRUE;
                                    22: 
                                        
                                        FB_Bacnet.StartStopCommand_085.bEnWrite := TRUE;
                                        FB_Bacnet.StartStopCommand_085.bVal := TRUE;
                                    23: 
                                        
                                        FB_Bacnet.StartStopCommand_225.bEnWrite := TRUE;
                                        FB_Bacnet.StartStopCommand_225.bVal := TRUE;
                                END_CASE
                            END_IF
                        END_FOR
                    END_IF
                    // Schedule Unit OFF
                    IF wSchedWDHourEndF37_ = currH AND wSchedWDMinEndF37_ = currM AND NOT bUnitTriggered THEN
                        bUnitTriggered := TRUE;
                        FOR i := 1 TO 23 DO
                            // Send command unit OFF
                            IF bUnitF37_[i] THEN 
                                CASE i OF
                                    1: 
                                        
                                        FB_Bacnet.StartStopCommand_064.bEnWrite := TRUE;
                                        FB_Bacnet.StartStopCommand_064.bVal := FALSE;
                                    2: 
                                        
                                        FB_Bacnet.StartStopCommand_065.bEnWrite := TRUE;
                                        FB_Bacnet.StartStopCommand_065.bVal := FALSE;
                                    3: 
                                        
                                        FB_Bacnet.StartStopCommand_066.bEnWrite := TRUE;
                                        FB_Bacnet.StartStopCommand_066.bVal := FALSE;
                                    4: 
                                        
                                        FB_Bacnet.StartStopCommand_067.bEnWrite := TRUE;
                                        FB_Bacnet.StartStopCommand_067.bVal := FALSE;
                                    5: 
                                        
                                        FB_Bacnet.StartStopCommand_068.bEnWrite := TRUE;
                                        FB_Bacnet.StartStopCommand_068.bVal := FALSE;
                                    6: 
                                        
                                        FB_Bacnet.StartStopCommand_069.bEnWrite := TRUE;
                                        FB_Bacnet.StartStopCommand_069.bVal := FALSE;
                                    7: 
                                        
                                        FB_Bacnet.StartStopCommand_070.bEnWrite := TRUE;
                                        FB_Bacnet.StartStopCommand_070.bVal := FALSE;
                                    8: 
                                        
                                        FB_Bacnet.StartStopCommand_071.bEnWrite := TRUE;
                                        FB_Bacnet.StartStopCommand_071.bVal := FALSE;
                                    9: 
                                        
                                        FB_Bacnet.StartStopCommand_072.bEnWrite := TRUE;
                                        FB_Bacnet.StartStopCommand_072.bVal := FALSE;
                                    10: 
                                        
                                        FB_Bacnet.StartStopCommand_073.bEnWrite := TRUE;
                                        FB_Bacnet.StartStopCommand_073.bVal := FALSE;
                                    11: 
                                        
                                        FB_Bacnet.StartStopCommand_074.bEnWrite := TRUE;
                                        FB_Bacnet.StartStopCommand_074.bVal := FALSE;
                                    12: 
                                        
                                        FB_Bacnet.StartStopCommand_075.bEnWrite := TRUE;
                                        FB_Bacnet.StartStopCommand_075.bVal := FALSE;
                                    13: 
                                        
                                        FB_Bacnet.StartStopCommand_076.bEnWrite := TRUE;
                                        FB_Bacnet.StartStopCommand_076.bVal := FALSE;
                                    14: 
                                        
                                        FB_Bacnet.StartStopCommand_077.bEnWrite := TRUE;
                                        FB_Bacnet.StartStopCommand_077.bVal := FALSE;
                                    15: 
                                        
                                        FB_Bacnet.StartStopCommand_078.bEnWrite := TRUE;
                                        FB_Bacnet.StartStopCommand_078.bVal := FALSE;
                                    16: 
                                        
                                        FB_Bacnet.StartStopCommand_079.bEnWrite := TRUE;
                                        FB_Bacnet.StartStopCommand_079.bVal := FALSE;
                                    17: 
                                        
                                        FB_Bacnet.StartStopCommand_080.bEnWrite := TRUE;
                                        FB_Bacnet.StartStopCommand_080.bVal := FALSE;
                                    18: 
                                        
                                        FB_Bacnet.StartStopCommand_081.bEnWrite := TRUE;
                                        FB_Bacnet.StartStopCommand_081.bVal := FALSE;
                                    19: 
                                        
                                        FB_Bacnet.StartStopCommand_082.bEnWrite := TRUE;
                                        FB_Bacnet.StartStopCommand_082.bVal := FALSE;
                                    20: 
                                        
                                        FB_Bacnet.StartStopCommand_083.bEnWrite := TRUE;
                                        FB_Bacnet.StartStopCommand_083.bVal := FALSE;
                                    21: 
                                        
                                        FB_Bacnet.StartStopCommand_084.bEnWrite := TRUE;
                                        FB_Bacnet.StartStopCommand_084.bVal := FALSE;
                                    22: 
                                        
                                        FB_Bacnet.StartStopCommand_085.bEnWrite := TRUE;
                                        FB_Bacnet.StartStopCommand_085.bVal := FALSE;
                                    23: 
                                        
                                        FB_Bacnet.StartStopCommand_225.bEnWrite := TRUE;
                                        FB_Bacnet.StartStopCommand_225.bVal := FALSE;
                                END_CASE
                            END_IF
                        END_FOR
                    END_IF
                END_IF
            END_IF

            // Weekend schedule
            IF currD = 0 OR currD = 6 THEN
                IF (wSchedWEHourStartF37_ <> wSchedWEHourEndF37_ OR wSchedWEMinStartF37_ <> wSchedWEMinEndF37_) THEN
                    // Schedule Unit ON
                    IF wSchedWEHourStartF37_ = currH AND wSchedWEMinStartF37_ = currM AND NOT bUnitTriggered THEN
                        bUnitTriggered := TRUE;
                        FOR i := 1 TO 23 DO
                            // Send command unit ON
                            IF bUnitF37_[i] THEN 
                                CASE i OF
                                    1: 
                                        
                                        FB_Bacnet.StartStopCommand_064.bEnWrite := TRUE;
                                        FB_Bacnet.StartStopCommand_064.bVal := TRUE;
                                    2: 
                                        
                                        FB_Bacnet.StartStopCommand_065.bEnWrite := TRUE;
                                        FB_Bacnet.StartStopCommand_065.bVal := TRUE;
                                    3: 
                                        
                                        FB_Bacnet.StartStopCommand_066.bEnWrite := TRUE;
                                        FB_Bacnet.StartStopCommand_066.bVal := TRUE;
                                    4: 
                                        
                                        FB_Bacnet.StartStopCommand_067.bEnWrite := TRUE;
                                        FB_Bacnet.StartStopCommand_067.bVal := TRUE;
                                    5: 
                                        
                                        FB_Bacnet.StartStopCommand_068.bEnWrite := TRUE;
                                        FB_Bacnet.StartStopCommand_068.bVal := TRUE;
                                    6: 
                                        
                                        FB_Bacnet.StartStopCommand_069.bEnWrite := TRUE;
                                        FB_Bacnet.StartStopCommand_069.bVal := TRUE;
                                    7: 
                                        
                                        FB_Bacnet.StartStopCommand_070.bEnWrite := TRUE;
                                        FB_Bacnet.StartStopCommand_070.bVal := TRUE;
                                    8: 
                                        
                                        FB_Bacnet.StartStopCommand_071.bEnWrite := TRUE;
                                        FB_Bacnet.StartStopCommand_071.bVal := TRUE;
                                    9: 
                                        
                                        FB_Bacnet.StartStopCommand_072.bEnWrite := TRUE;
                                        FB_Bacnet.StartStopCommand_072.bVal := TRUE;
                                    10: 
                                        
                                        FB_Bacnet.StartStopCommand_073.bEnWrite := TRUE;
                                        FB_Bacnet.StartStopCommand_073.bVal := TRUE;
                                    11: 
                                        
                                        FB_Bacnet.StartStopCommand_074.bEnWrite := TRUE;
                                        FB_Bacnet.StartStopCommand_074.bVal := TRUE;
                                    12: 
                                        
                                        FB_Bacnet.StartStopCommand_075.bEnWrite := TRUE;
                                        FB_Bacnet.StartStopCommand_075.bVal := TRUE;
                                    13: 
                                        
                                        FB_Bacnet.StartStopCommand_076.bEnWrite := TRUE;
                                        FB_Bacnet.StartStopCommand_076.bVal := TRUE;
                                    14: 
                                        
                                        FB_Bacnet.StartStopCommand_077.bEnWrite := TRUE;
                                        FB_Bacnet.StartStopCommand_077.bVal := TRUE;
                                    15: 
                                        
                                        FB_Bacnet.StartStopCommand_078.bEnWrite := TRUE;
                                        FB_Bacnet.StartStopCommand_078.bVal := TRUE;
                                    16: 
                                        
                                        FB_Bacnet.StartStopCommand_079.bEnWrite := TRUE;
                                        FB_Bacnet.StartStopCommand_079.bVal := TRUE;
                                    17: 
                                        
                                        FB_Bacnet.StartStopCommand_080.bEnWrite := TRUE;
                                        FB_Bacnet.StartStopCommand_080.bVal := TRUE;
                                    18: 
                                        
                                        FB_Bacnet.StartStopCommand_081.bEnWrite := TRUE;
                                        FB_Bacnet.StartStopCommand_081.bVal := TRUE;
                                    19: 
                                        
                                        FB_Bacnet.StartStopCommand_082.bEnWrite := TRUE;
                                        FB_Bacnet.StartStopCommand_082.bVal := TRUE;
                                    20: 
                                        
                                        FB_Bacnet.StartStopCommand_083.bEnWrite := TRUE;
                                        FB_Bacnet.StartStopCommand_083.bVal := TRUE;
                                    21: 
                                        
                                        FB_Bacnet.StartStopCommand_084.bEnWrite := TRUE;
                                        FB_Bacnet.StartStopCommand_084.bVal := TRUE;
                                    22: 
                                        
                                        FB_Bacnet.StartStopCommand_085.bEnWrite := TRUE;
                                        FB_Bacnet.StartStopCommand_085.bVal := TRUE;
                                    23: 
                                        
                                        FB_Bacnet.StartStopCommand_225.bEnWrite := TRUE;
                                        FB_Bacnet.StartStopCommand_225.bVal := TRUE;
                                END_CASE
                            END_IF
                        END_FOR        
                    END_IF
                    // Schedule Unit OFF
                    IF wSchedWEHourEndF37_ = currH AND wSchedWEMinEndF37_ = currM AND NOT bUnitTriggered THEN
                        bUnitTriggered := TRUE;
                        FOR i := 1 TO 23 DO
                            // Send command unit OFF
                            IF bUnitF37_[i] THEN 
                                CASE i OF
                                    1: 
                                        
                                        FB_Bacnet.StartStopCommand_064.bEnWrite := TRUE;
                                        FB_Bacnet.StartStopCommand_064.bVal := FALSE;
                                    2: 
                                        
                                        FB_Bacnet.StartStopCommand_065.bEnWrite := TRUE;
                                        FB_Bacnet.StartStopCommand_065.bVal := FALSE;
                                    3: 
                                        
                                        FB_Bacnet.StartStopCommand_066.bEnWrite := TRUE;
                                        FB_Bacnet.StartStopCommand_066.bVal := FALSE;
                                    4: 
                                        
                                        FB_Bacnet.StartStopCommand_067.bEnWrite := TRUE;
                                        FB_Bacnet.StartStopCommand_067.bVal := FALSE;
                                    5: 
                                        
                                        FB_Bacnet.StartStopCommand_068.bEnWrite := TRUE;
                                        FB_Bacnet.StartStopCommand_068.bVal := FALSE;
                                    6: 
                                        
                                        FB_Bacnet.StartStopCommand_069.bEnWrite := TRUE;
                                        FB_Bacnet.StartStopCommand_069.bVal := FALSE;
                                    7: 
                                        
                                        FB_Bacnet.StartStopCommand_070.bEnWrite := TRUE;
                                        FB_Bacnet.StartStopCommand_070.bVal := FALSE;
                                    8: 
                                        
                                        FB_Bacnet.StartStopCommand_071.bEnWrite := TRUE;
                                        FB_Bacnet.StartStopCommand_071.bVal := FALSE;
                                    9: 
                                        
                                        FB_Bacnet.StartStopCommand_072.bEnWrite := TRUE;
                                        FB_Bacnet.StartStopCommand_072.bVal := FALSE;
                                    10: 
                                        
                                        FB_Bacnet.StartStopCommand_073.bEnWrite := TRUE;
                                        FB_Bacnet.StartStopCommand_073.bVal := FALSE;
                                    11: 
                                        
                                        FB_Bacnet.StartStopCommand_074.bEnWrite := TRUE;
                                        FB_Bacnet.StartStopCommand_074.bVal := FALSE;
                                    12: 
                                        
                                        FB_Bacnet.StartStopCommand_075.bEnWrite := TRUE;
                                        FB_Bacnet.StartStopCommand_075.bVal := FALSE;
                                    13: 
                                        
                                        FB_Bacnet.StartStopCommand_076.bEnWrite := TRUE;
                                        FB_Bacnet.StartStopCommand_076.bVal := FALSE;
                                    14: 
                                        
                                        FB_Bacnet.StartStopCommand_077.bEnWrite := TRUE;
                                        FB_Bacnet.StartStopCommand_077.bVal := FALSE;
                                    15: 
                                        
                                        FB_Bacnet.StartStopCommand_078.bEnWrite := TRUE;
                                        FB_Bacnet.StartStopCommand_078.bVal := FALSE;
                                    16: 
                                        
                                        FB_Bacnet.StartStopCommand_079.bEnWrite := TRUE;
                                        FB_Bacnet.StartStopCommand_079.bVal := FALSE;
                                    17: 
                                        
                                        FB_Bacnet.StartStopCommand_080.bEnWrite := TRUE;
                                        FB_Bacnet.StartStopCommand_080.bVal := FALSE;
                                    18: 
                                        
                                        FB_Bacnet.StartStopCommand_081.bEnWrite := TRUE;
                                        FB_Bacnet.StartStopCommand_081.bVal := FALSE;
                                    19: 
                                        
                                        FB_Bacnet.StartStopCommand_082.bEnWrite := TRUE;
                                        FB_Bacnet.StartStopCommand_082.bVal := FALSE;
                                    20: 
                                        
                                        FB_Bacnet.StartStopCommand_083.bEnWrite := TRUE;
                                        FB_Bacnet.StartStopCommand_083.bVal := FALSE;
                                    21: 
                                        
                                        FB_Bacnet.StartStopCommand_084.bEnWrite := TRUE;
                                        FB_Bacnet.StartStopCommand_084.bVal := FALSE;
                                    22: 
                                        
                                        FB_Bacnet.StartStopCommand_085.bEnWrite := TRUE;
                                        FB_Bacnet.StartStopCommand_085.bVal := FALSE;
                                    23: 
                                        
                                        FB_Bacnet.StartStopCommand_225.bEnWrite := TRUE;
                                        FB_Bacnet.StartStopCommand_225.bVal := FALSE;
                                END_CASE
                            END_IF
                        END_FOR
                    END_IF
                END_IF
            END_IF
        END_IF

END_FUNCTION_BLOCK

// ---- POUs/FB_Scheduler/FB_Scheduler_F38.TcPOU

      FUNCTION_BLOCK FB_Scheduler_F38
      VAR_INPUT
          currH : WORD;
          currM : WORD;
          currD : WORD;
      END_VAR
      VAR_IN_OUT
          FB_Bacnet : FB_BACnet_DAIKIN_MasterStation_III_No_9;
      END_VAR
      VAR
          i : INT;
          bUnitTriggered : BOOL := FALSE; // New flag to track execution
          prevMinute : WORD := 0;        // New variable to track the previous minute
      END_VAR
      VAR PERSISTENT
          //scheduler var
          bEnSchedF38_ : BOOL := FALSE;
          wSchedWDHourStartF38_ : WORD; 
          wSchedWDMinStartF38_ : WORD; 
          wSchedWEHourStartF38_ : WORD; 
          wSchedWEMinStartF38_ : WORD;
          wSchedWDHourEndF38_ : WORD;
          wSchedWDMinEndF38_ : WORD;
          wSchedWEHourEndF38_ : WORD;
          wSchedWEMinEndF38_ : WORD;
          //unit var
          bUnitF38_ : ARRAY [1..25] OF BOOL;
      END_VAR


        // Reset trigger flag at minute change or at the exact scheduled time
        IF currM <> prevMinute OR 
           (currH = wSchedWDHourStartF38_ AND currM = wSchedWDMinStartF38_) OR 
           (currH = wSchedWDHourEndF38_ AND currM = wSchedWDMinEndF38_) THEN
            bUnitTriggered := FALSE;
            prevMinute := currM;
        END_IF

        // Unit Schedule Enable
        IF bEnSchedF38_ THEN
            // Weekday schedule
            IF currD >= 1 AND currD <= 5 THEN
                IF (wSchedWDHourStartF38_ <> wSchedWDHourEndF38_ OR wSchedWDMinStartF38_ <> wSchedWDMinEndF38_) THEN
                    // Schedule Unit ON
                    IF wSchedWDHourStartF38_ = currH AND wSchedWDMinStartF38_ = currM AND NOT bUnitTriggered THEN
                        bUnitTriggered := TRUE;
                        FOR i := 1 TO 25 DO
                            // Send command unit ON
                            IF bUnitF38_[i] THEN 
                                CASE i OF
                                    1: 
                                        
                                        FB_Bacnet.StartStopCommand_128.bEnWrite := TRUE;
                                        FB_Bacnet.StartStopCommand_128.bVal := TRUE;
                                    2: 
                                        
                                        FB_Bacnet.StartStopCommand_129.bEnWrite := TRUE;
                                        FB_Bacnet.StartStopCommand_129.bVal := TRUE;
                                    3: 
                                        
                                        FB_Bacnet.StartStopCommand_130.bEnWrite := TRUE;
                                        FB_Bacnet.StartStopCommand_130.bVal := TRUE;
                                    4: 
                                        
                                        FB_Bacnet.StartStopCommand_131.bEnWrite := TRUE;
                                        FB_Bacnet.StartStopCommand_131.bVal := TRUE;
                                    5: 
                                        
                                        FB_Bacnet.StartStopCommand_132.bEnWrite := TRUE;
                                        FB_Bacnet.StartStopCommand_132.bVal := TRUE;
                                    6: 
                                        
                                        FB_Bacnet.StartStopCommand_133.bEnWrite := TRUE;
                                        FB_Bacnet.StartStopCommand_133.bVal := TRUE;
                                    7: 
                                        
                                        FB_Bacnet.StartStopCommand_134.bEnWrite := TRUE;
                                        FB_Bacnet.StartStopCommand_134.bVal := TRUE;
                                    8: 
                                        
                                        FB_Bacnet.StartStopCommand_135.bEnWrite := TRUE;
                                        FB_Bacnet.StartStopCommand_135.bVal := TRUE;
                                    9: 
                                        
                                        FB_Bacnet.StartStopCommand_136.bEnWrite := TRUE;
                                        FB_Bacnet.StartStopCommand_136.bVal := TRUE;
                                    10: 
                                        
                                        FB_Bacnet.StartStopCommand_137.bEnWrite := TRUE;
                                        FB_Bacnet.StartStopCommand_137.bVal := TRUE;
                                    11: 
                                        
                                        FB_Bacnet.StartStopCommand_138.bEnWrite := TRUE;
                                        FB_Bacnet.StartStopCommand_138.bVal := TRUE;
                                    12: 
                                        
                                        FB_Bacnet.StartStopCommand_139.bEnWrite := TRUE;
                                        FB_Bacnet.StartStopCommand_139.bVal := TRUE;
                                    13: 
                                        
                                        FB_Bacnet.StartStopCommand_140.bEnWrite := TRUE;
                                        FB_Bacnet.StartStopCommand_140.bVal := TRUE;
                                    14: 
                                        
                                        FB_Bacnet.StartStopCommand_141.bEnWrite := TRUE;
                                        FB_Bacnet.StartStopCommand_141.bVal := TRUE;
                                    15: 
                                        
                                        FB_Bacnet.StartStopCommand_142.bEnWrite := TRUE;
                                        FB_Bacnet.StartStopCommand_142.bVal := TRUE;
                                    16: 
                                        
